{attribute 'Tc2GvlVarNames'}
VAR_CONFIG
END_VAR

(* stored: Version 1.1.0.1, ProductVersion 3.1.4022.9
   GVL Variable_Configuration: Id {449d693c-1c41-4961-ad41-92587592bc85} *)
